(* CODESYS project TREINO_PROVA.project

Project tree, tasks and I/O mapping:
  Device : CODESYS Control Win V3, 3S - Smart Software Solutions GmbH, order no. 305021, version 3.5.11.30
    application Application
      libraries: Standard, * (System)
      task MainTask (cyclic, interval t#20ms, priority 1) calls PLC_PRG
      program PLC_PRG [LD]
*)

// Device/Application/PLC_PRG
PROGRAM PLC_PRG
VAR
	STIR : BOOL;  //motor (220Vac monofásico ON/OFF)
    EST  : BOOL;  // Uma esteira com o material sólido é controlada por um motor(220Vac monofásico ON/OFF)
    MV1  : BOOL;  // A válvula magnética (NF 220Vac) controla a entrada de água no tanque
    MV2  : BOOL;  // (NF 220Vac) controla a saída de produto do tanque
    LT1  : BOOL; // sensor de níveL (24Vdc NA) que quando detectar material (líquido ou sólido) se tornam ativos
    LT2  : BOOL; // sensor de níveL (24Vdc NA) que quando detectar material (líquido ou sólido) se tornam ativos
    LT3  : BOOL; // sensor de níveL (24Vdc NA) que quando detectar material (líquido ou sólido) se tornam ativos
    START: BOOL; // para ligar o sistema
	STOP : BOOL; // para desligar o sistema
	P1: BOOL;
	P2: BOOL;
	P3: BOOL;
	TOF_1: TOF;
	ET1: TIME;
	TON_1: TON;
	ET2: TIME;
	AUX: BOOL;
END_VAR
VAR // added by the converter: edge detectors and wires of the graphical bodies
    _w1 : BOOL;
    _rt1 : R_TRIG;
    _ft1 : F_TRIG;
END_VAR

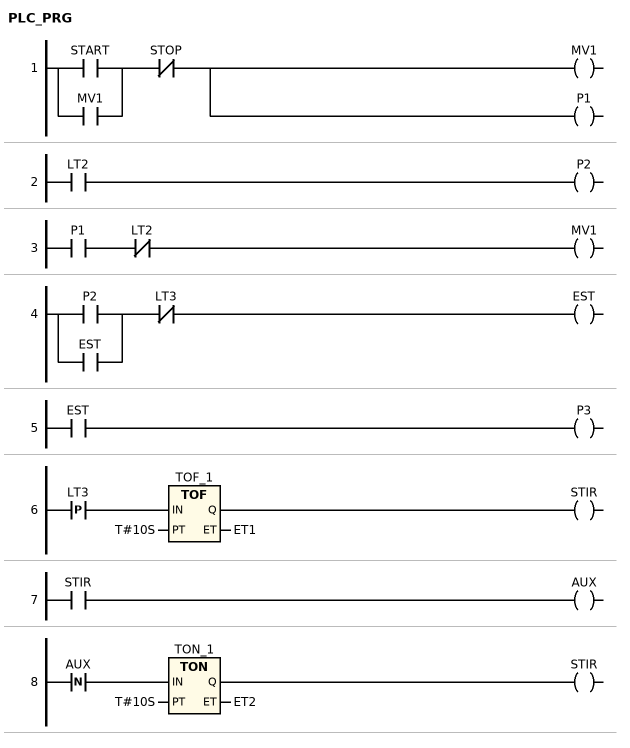
// NETWORK 1
_w1 := (START OR MV1) AND NOT STOP;
MV1 := _w1;
P1 := _w1;

// NETWORK 2
P2 := LT2;

// NETWORK 3
MV1 := P1 AND NOT LT2;

// NETWORK 4
EST := (P2 OR EST) AND NOT LT3;

// NETWORK 5
P3 := EST;

// NETWORK 6
_rt1(CLK := LT3);
TOF_1(IN := _rt1.Q, PT := T#10S, ET => ET1); // TOF
STIR := TOF_1.Q;

// NETWORK 7
AUX := STIR;

// NETWORK 8
_ft1(CLK := AUX);
TON_1(IN := _ft1.Q, PT := T#10S, ET => ET2); // TON
STIR := TON_1.Q;

END_PROGRAM
